FUNCTION_BLOCK TcoTixonPickStepSeparatorTask EXTENDS TcoTixonFeedingTask
VAR_IN_OUT
    inoConfig : TcoTixonPickStep_Config_v_1_x_x;
    inoControl : TcoTixonPickStep_Control_v_1_x_x;
    inoStatus : TcoTixonPickStep_Status_v_1_x_x;
END_VAR
VAR
    _componentReady : BOOL;
END_VAR

IF Execute() THEN
    IF _progress = 0 THEN
        IF NOT __ISVALIDREF(inoControl) THEN
            _varInfo := __VARINFO(inoControl);
            Messenger.Programming(_sb.Clear().Append('<#Invalid reference: #>').Append(_varInfo.Symbol).ToString()).Pin();
        ELSIF NOT __ISVALIDREF(inoConfig) THEN
            _varInfo := __VARINFO(inoConfig);
            Messenger.Programming(_sb.Clear().Append('<#Invalid reference: #>').Append(_varInfo.Symbol).ToString()).Pin();
        ELSIF NOT __ISVALIDREF(inoStatus) THEN
            _varInfo := __VARINFO(inoStatus);
            Messenger.Programming(_sb.Clear().Append('<#Invalid reference: #>').Append(_varInfo.Symbol).ToString()).Pin();
        ELSIF NOT inoStatus.ControllerInAuto THEN
            _varInfo := __VARINFO(inoStatus.ControllerInAuto);
            Messenger.Warning(_sb.Clear().Append('<#Tixon control system not in auto #>').Append(_varInfo.Symbol).ToString());
        ELSIF NOT inoConfig.SeparatorActive THEN
            _progress := 4;
        ELSE
            _progress := _progress + 1;
        END_IF
    END_IF

    IF _progress = 1 THEN
        inoControl.SepareComponent := FALSE;
        _varInfo := __VARINFO(inoStatus.SeparatorHomePos);

        THIS^.Messenger.OnCondition(_infoTimer.Q AND NOT inoStatus.SeparatorHomePos)
            .Warning(_sb.Clear().Append('<#Waiting for #>').Append(_varInfo.Symbol).ToString());

        IF inoStatus.SeparatorHomePos THEN
            _progress := _progress + 1;
            _timer(In := FALSE);
        END_IF;
    END_IF;

    IF _progress = 2 THEN
        Messenger.Debug('<#Waiting for component in  separator#>');
        _timer(IN := inoStatus.SeparatorPresent, Pt := inoConfig.TimeToComponentInSeparator);

        IF _timer.Q THEN
            _progress := _progress + 1;
            _timer(In := FALSE);
        END_IF
    END_IF;

    IF _progress = 3 THEN
        inoControl.SepareComponent := TRUE;
        _varInfo := __VARINFO(inoStatus.SeparatorWorkPos);

        THIS^.Messenger.OnCondition(_infoTimer.Q AND NOT inoStatus.SeparatorWorkPos)
            .Warning(_sb.Clear().Append('<#Waiting for #>').Append(_varInfo.Symbol).ToString());

        IF inoStatus.SeparatorWorkPos THEN
            _progress := _progress + 1;
            _timer(In := FALSE);
        END_IF;
    END_IF;

    IF _progress = 4 THEN
        Messenger.Debug('<#Waiting for component in Pick position#>');
        _timer(IN := inoStatus.SeparatorPresent, Pt := inoConfig.TimeToComponentOutSeparator);

        IF inoStatus.SeparatorPresent THEN
            _progress := _progress + 1;
            _timer(In := FALSE);
        END_IF
    END_IF;

    IF _progress = 5 THEN
        _componentReady := TRUE;
        THIS^.DoneWhen(TRUE);
    END_IF;

    CallTimers(TRUE);
    THIS^.ThrowWhen(_errorTimer.Q);
END_IF

inoStatus.ComponentReady := _componentReady;

IF THIS^.Error AND NOT _errorMessage.Pinned THEN
    THIS^.Restore();
END_IF

PROPERTY PUBLIC ComponentReady : bool
GET
ComponentReady := _componentReady;
END_GET
END_PROPERTY

(*~
    <docu>
        <summary>
            Executes when task is aborted.
        </summary>
    </docu>
~*)
METHOD PROTECTED OnAbort
IF __ISVALIDREF(inoStatus) THEN
    THIS^.inoStatus.ActionDescription := '<#Separator task  was aborted.#>';
END_IF;
END_METHOD

(*~
    <docu>
        <summary>
            Executes when task reaches the ```Done``` state .
        </summary>
    </docu>
~*)
METHOD PROTECTED OnDone
IF __ISVALIDREF(inoStatus) THEN
    THIS^.inoStatus.ActionDescription := '<#Separator task  finished successfully.#>';
END_IF;

_progress := 0;

IF AutoRestore THEN
    Restore();
END_IF
END_METHOD

METHOD PROTECTED OnError
VAR
    description : STRING;
END_VAR
description := '<#Separator task finished with error.#>';
_componentReady := false;

IF __ISVALIDREF(inoStatus) THEN
    THIS^.inoStatus.ActionDescription := description;
END_IF;

THIS^._errorMessage.Error(_sb.Clear().Append(description).Append(' To restore acknowledge this alarm.').ToString()).Pin();
END_METHOD

METHOD PROTECTED OnStart
IF __ISVALIDREF(inoStatus) THEN
    THIS^.inoStatus.ActionDescription := '<#Separator task started.#>';
END_IF;

_componentReady := false;
CallTimers(FALSE);
END_METHOD

(*~
    <docu>
        <summary>
            Restores this instance to the Ready state. Can be called explicitly or from within one of the restore mechanisms.
            <para>
                See also <see cref="PlcDocu.TcoCore.TcoTask.AutoRestorable()"/>
            </para>
        </summary>
    </docu>
~*)
METHOD Restore : ITcoRestorable
SUPER^.Restore();
_componentReady := false;
END_METHOD

END_FUNCTION_BLOCK

(* stored: Version 1.1.0.1, ProductVersion 3.1.4024.12
   POU TcoTixonPickStepSeparatorTask: Id {ac76e352-eb60-01d0-2737-d7abcd936e64}, SpecialFunc None
   Property ComponentReady: Id {ed1f4a44-d784-0daa-3bc2-d6633a9627a9}
   Get Get: Id {d65a8e30-4c52-0919-05cc-92b421a6e1b3}
   Method OnAbort: Id {14e4fd0d-7e5f-0f46-09ad-ba1c3ee32096}
   Method OnDone: Id {7340e635-1e74-0fae-266f-0393008e2807}
   Method OnError: Id {ab114dd6-4d9a-0bce-3f27-68e80c659893}
   Method OnStart: Id {d75015c0-5a38-0c5d-369f-5619dd147cf7}
   Method Restore: Id {5f4f8652-2f9b-0082-3967-b05ac2c49250} *)
